// TIA Portal project "PalettizerKontrolUygulamasi" (V17)
// Vorlageprojekt für das Buch mit Zielsystem S7-1200

(* hardware
DEVICE "S7-1200-Station_1"  S7-1200 Station
   slot 0: "Baugruppenträger_0"  Rack  V1.0
   slot 1: "PLC_1"  CPU 1211C DC/DC/DC  6ES7 211-1AE40-0XB0  V4.1
*)

// ===== PLC "PLC_1"  CPU 1211C DC/DC/DC =====

VAR_GLOBAL   // PLC tag table "Standard-Variablentabelle"
   "Tag_1" AT %A0.0 : Bool;
   "Tag_2" AT %E0.0 : Bool;
   "Tag_3" AT %E0.1 : Bool;
   "AUTO" AT %I1.4 : Bool;
   "START" AT %I1.0 : Bool;
   "START LIGHT" AT %Q1.5 : Bool;
   "WARNİNG LIGHT" AT %Q1.4 : Bool;
   "BOX FEEDER" AT %Q0.6 : Bool;
   "LOAD BELT" AT %Q1.1 : Bool;
   "STOP LIGHT" AT %Q1.7 : Bool;
   "COUNTER" AT %QD30 : DWord;
   "BOX AT ENTRY" AT %I0.3 : Bool;
   "Tag_6" AT %M0.0 : Bool;
   "Tag_4" AT %QD40 : DWord;
   "Tag_5" AT %M10.0 : Bool;
   "Tag_7" AT %M10.1 : Bool;
   "ELEVATOR DOWN" AT %Q0.5 : Bool;
   "PUSH" AT %Q1.0 : Bool;
   "PUSHER LİMİT" AT %I0.4 : Bool;
   "Tag_9" AT %M0.3 : Bool;
   "Tag_8" AT %M10.6 : Bool;
   "ELEVATOR UP" AT %Q0.4 : Bool;
   "EXİT CONVEYOR" AT %Q0.2 : Bool;
   "MOVE TO LİMİT" AT %Q0.3 : Bool;
   "Tag_10" AT %M0.4 : Bool;
   "CLAMP" AT %Q1.2 : Bool;
   "Tag_12" AT %M10.2 : Bool;
   "CLAMPED" AT %I0.6 : Bool;
   "OPEN PLATE" AT %Q1.3 : Bool;
   "Tag_14" AT %M10.3 : Bool;
   "Tag_11" AT %M10.5 : Bool;
   "PLATE LİMİT" AT %I0.5 : Bool;
   "Tag_15" AT %M0.7 : Bool;
   "Tag_13" AT %M10.4 : Bool;
   "TURN" AT %Q0.7 : Bool;
   "Tag_16" AT %M1.1 : Bool;
   "Tag_17" AT %M10.7 : Bool;
   "Tag_18" AT %M1.2 : Bool;
   "Tag_19" AT %M11.0 : Bool;
   "Tag_20" AT %M11.1 : Bool;
   "Tag_21" AT %M1.3 : Bool;
   "Tag_22" AT %QD50 : DInt;
END_VAR

// folder: System blocks/Program resources

DATA_BLOCK "IEC_Timer_0_DB"   // DB1
{ S7_Optimized_Access := 'TRUE' }
AUTHOR : Simatic
FAMILY : IEC
NAME : IEC_TMR
VERSION : 1.0
// stored: InstanceOfName IEC_TIMER
"IEC_TIMER"
BEGIN
END_DATA_BLOCK

DATA_BLOCK "IEC_Timer_0_DB_1"   // DB2
{ S7_Optimized_Access := 'TRUE' }
AUTHOR : Simatic
FAMILY : IEC
NAME : IEC_TMR
VERSION : 1.0
// stored: InstanceOfName IEC_TIMER
"IEC_TIMER"
BEGIN
END_DATA_BLOCK

DATA_BLOCK "IEC_Timer_0_DB_2"   // DB3
{ S7_Optimized_Access := 'TRUE' }
AUTHOR : Simatic
FAMILY : IEC
NAME : IEC_TMR
VERSION : 1.0
// stored: InstanceOfName IEC_TIMER
"IEC_TIMER"
BEGIN
END_DATA_BLOCK

DATA_BLOCK "IEC_Timer_0_DB_3"   // DB4
{ S7_Optimized_Access := 'TRUE' }
AUTHOR : Simatic
FAMILY : IEC
NAME : IEC_TMR
VERSION : 1.0
// stored: InstanceOfName IEC_TIMER
"IEC_TIMER"
BEGIN
END_DATA_BLOCK

// folder: (top level)

FUNCTION "MHJ-PLC-Lab-Function-S71200" : Void   // FC9000, SCL
{ S7_Optimized_Access := 'TRUE' }
VERSION : 0.1
   VAR_TEMP
      rdTimeReturn : Int;
      outputTime : DTL;
      SyncVal : Byte;
      forVal : Int;
      forVal_2 : Int;
      Value : Byte;
   END_VAR
   VAR CONSTANT
      CompVal : Byte := 16#34;
      Value_01 : Byte := 16#11;
      Value_01_DW : DWord := 16#A165_D992;
      Value_02_DW : DWord := 16#58BE_4401;
   END_VAR
BEGIN

   #Value:=PEEK(area := 16#82,
        dbNumber := 0,
        byteOffset := 511);
   #Value := #Value + 1;

   POKE(area := 16#82,
        dbNumber := 0,
        byteOffset := 511,
        value := #Value);

   POKE(area:=16#81,
        dbNumber:=0,
        byteOffset:=1016,
        value:=#Value_01_DW);
   POKE(area := 16#81,
        dbNumber := 0,
        byteOffset := 1020,
        value := #Value_02_DW);

   POKE(area := 16#81,
        dbNumber := 0,
        byteOffset := 511,
        value := B#16#00);

   FOR #forVal := 0 TO 120 DO
       FOR #forVal_2:=0 TO 10 DO
           #rdTimeReturn:=RD_SYS_T(#outputTime);
           #rdTimeReturn := WR_SYS_T(#outputTime);
           #rdTimeReturn := RD_SYS_T(#outputTime);
           #rdTimeReturn := WR_SYS_T(#outputTime);
       END_FOR;
       #SyncVal:= PEEK(area := 16#81,
                      dbNumber := 0,
                      byteOffset := 511);
       IF #SyncVal = #CompVal THEN
          GOTO M_1;
       END_IF;
   END_FOR;
   RETURN;

   M_1:
   POKE(area := 16#81,
        dbNumber := 0,
        byteOffset := 511,
        value := B#16#0);
END_FUNCTION

ORGANIZATION_BLOCK "Main"   // OB1, LAD, ProgramCycle
TITLE = "Main Program Sweep (Cycle)"
{ S7_Optimized_Access := 'TRUE' }
VERSION : 0.1
   VAR_INPUT
      Initial_Call : Bool;   // Initial call of this OB
      Remanence : Bool;   // =True, if remanent data are available
   END_VAR
   VAR_TEMP   // added for the SCL form of the ladder/FBD networks
      _w1 : Bool;
      _w2 : Bool;
      _w3 : Bool;
      _w4 : Bool;
      _w5 : Bool;
      _w6 : Bool;
      _w7 : Bool;
      _w8 : Bool;
      _w9 : Bool;
      _w10 : Bool;
      _w11 : Bool;
      _w12 : Bool;
      _w13 : Bool;
   END_VAR
BEGIN

REGION Network 1: Konnektierungsbaustein für PLC-Lab
   // Im Netzwerk 1 wird der Konnektierungsbaustein für PLC-Lab aufgerufen.
   // Dieser Aufruf darf nicht entfernt werden!
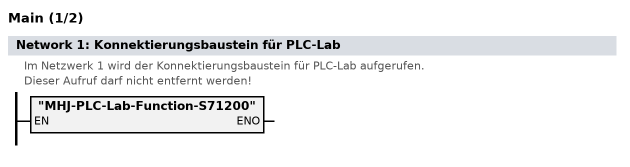
   RUNG wire#powerrail
      "MHJ-PLC-Lab-Function-S71200"()
   END_RUNG
   // the same network as SCL:
   "MHJ-PLC-Lab-Function-S71200"();
END_REGION

REGION Network 2: Ihr Programm
   // Schreiben Sie ab Netzwerk 2 Ihr Programm
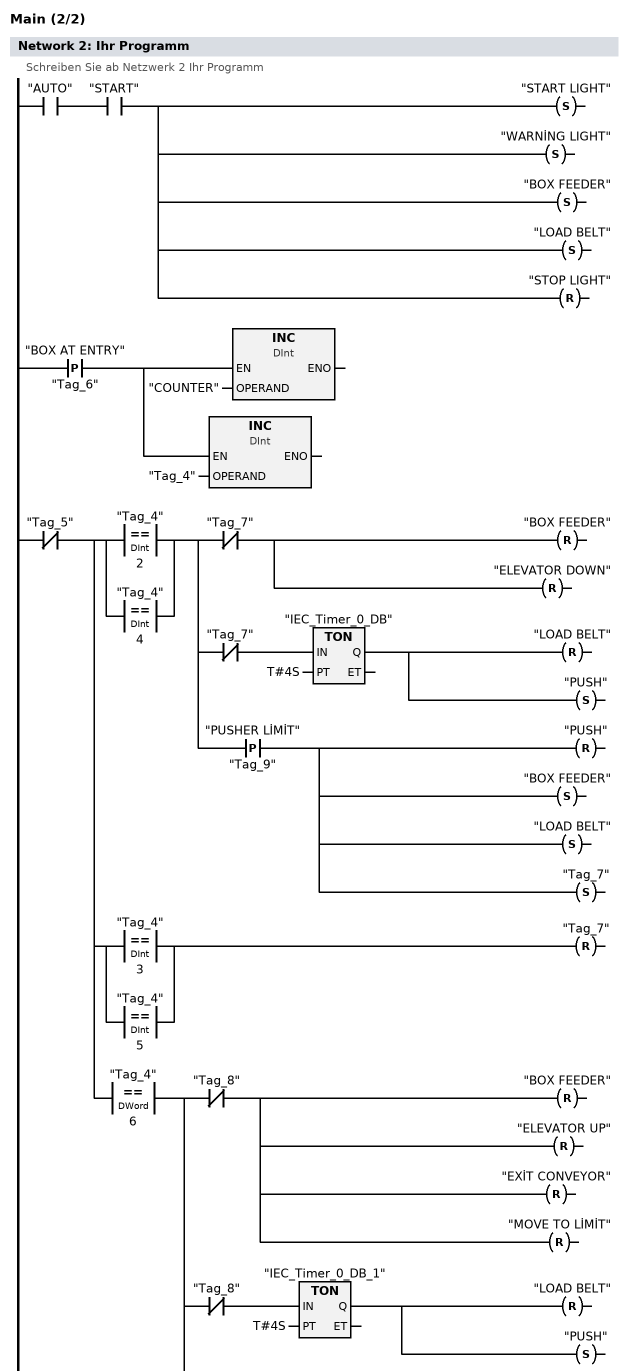
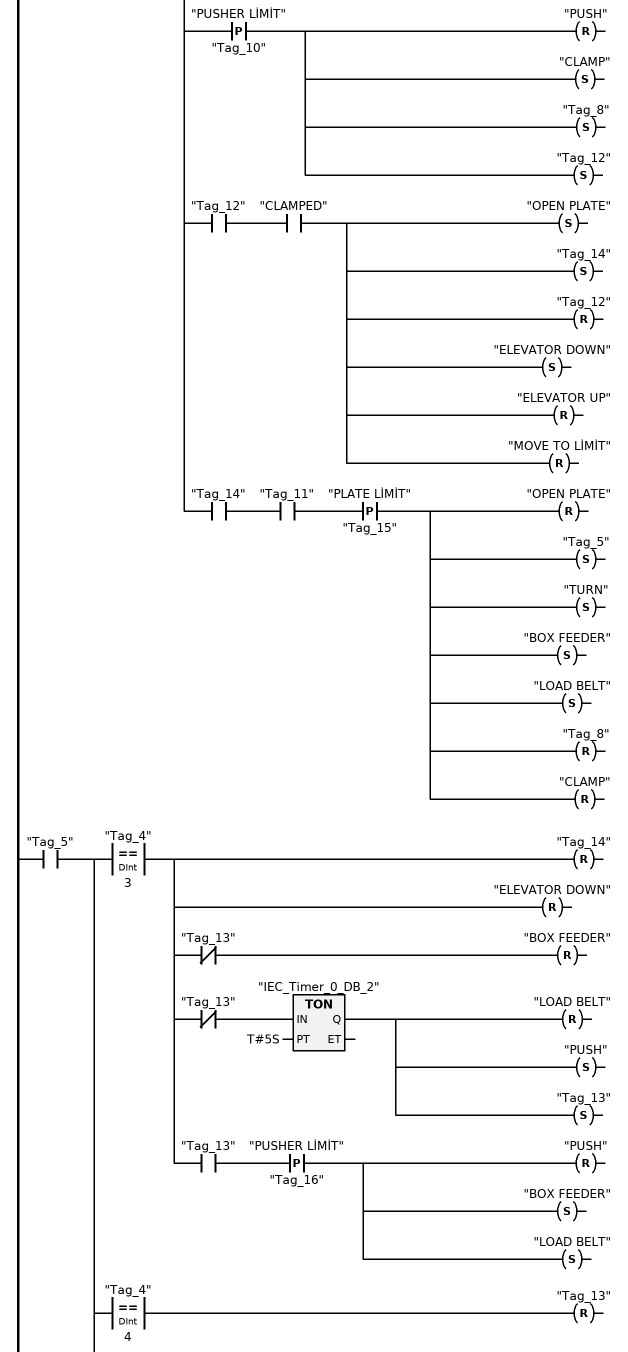
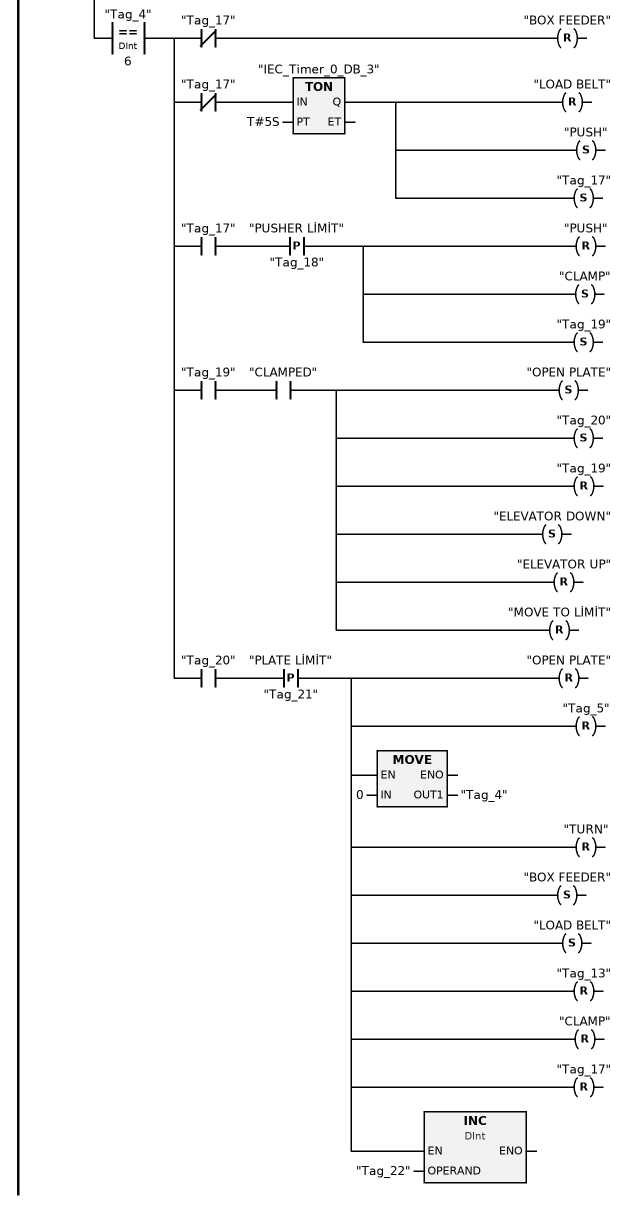
   IF "AUTO" AND "START" THEN
       "START LIGHT" := TRUE;
       "WARNİNG LIGHT" := TRUE;
       "BOX FEEDER" := TRUE;
       "LOAD BELT" := TRUE;
       "STOP LIGHT" := FALSE;
   END_IF;
   #_w1 := "BOX AT ENTRY" AND NOT "Tag_6";   // rising edge of "BOX AT ENTRY"
   "Tag_6" := "BOX AT ENTRY";
   IF #_w1 THEN
       "COUNTER" := "COUNTER" + 1;
       "Tag_4" := "Tag_4" + 1;
   END_IF;
   #_w2 := NOT "Tag_5" AND (("Tag_4" = 2) OR ("Tag_4" = 4));
   IF #_w2 AND NOT "Tag_7" THEN
       "BOX FEEDER" := FALSE;
       "ELEVATOR DOWN" := FALSE;
   END_IF;
   "IEC_Timer_0_DB".TON(IN := #_w2 AND NOT "Tag_7", PT := T#4S);
   IF "IEC_Timer_0_DB".Q THEN
       "LOAD BELT" := FALSE;
       "PUSH" := TRUE;
   END_IF;
   #_w3 := #_w2 AND "PUSHER LİMİT" AND NOT "Tag_9";   // rising edge of "PUSHER LİMİT"
   "Tag_9" := "PUSHER LİMİT";
   IF #_w3 THEN
       "PUSH" := FALSE;
       "BOX FEEDER" := TRUE;
       "LOAD BELT" := TRUE;
       "Tag_7" := TRUE;
   END_IF;
   IF NOT "Tag_5" AND (("Tag_4" = 3) OR ("Tag_4" = 5)) THEN "Tag_7" := FALSE; END_IF;
   #_w4 := NOT "Tag_5" AND ("Tag_4" = 6);
   IF #_w4 AND NOT "Tag_8" THEN
       "BOX FEEDER" := FALSE;
       "ELEVATOR UP" := FALSE;
       "EXİT CONVEYOR" := FALSE;
       "MOVE TO LİMİT" := FALSE;
   END_IF;
   "IEC_Timer_0_DB_1".TON(IN := #_w4 AND NOT "Tag_8", PT := T#4S);
   IF "IEC_Timer_0_DB_1".Q THEN
       "LOAD BELT" := FALSE;
       "PUSH" := TRUE;
   END_IF;
   #_w5 := #_w4 AND "PUSHER LİMİT" AND NOT "Tag_10";   // rising edge of "PUSHER LİMİT"
   "Tag_10" := "PUSHER LİMİT";
   IF #_w5 THEN
       "PUSH" := FALSE;
       "CLAMP" := TRUE;
       "Tag_8" := TRUE;
       "Tag_12" := TRUE;
   END_IF;
   IF #_w4 AND "Tag_12" AND "CLAMPED" THEN
       "OPEN PLATE" := TRUE;
       "Tag_14" := TRUE;
   END_IF;
   #_w6 := #_w4 AND "Tag_12" AND "CLAMPED";
   IF #_w6 THEN
       "Tag_12" := FALSE;
       "ELEVATOR DOWN" := TRUE;
       "ELEVATOR UP" := FALSE;
       "MOVE TO LİMİT" := FALSE;
   END_IF;
   #_w7 := #_w4 AND "Tag_14" AND "Tag_11" AND "PLATE LİMİT" AND NOT "Tag_15";   // rising edge of "PLATE LİMİT"
   "Tag_15" := "PLATE LİMİT";
   IF #_w7 THEN
       "OPEN PLATE" := FALSE;
       "Tag_5" := TRUE;
       "TURN" := TRUE;
       "BOX FEEDER" := TRUE;
       "LOAD BELT" := TRUE;
       "Tag_8" := FALSE;
       "CLAMP" := FALSE;
   END_IF;
   #_w8 := "Tag_5" AND ("Tag_4" = 3);
   IF #_w8 THEN
       "Tag_14" := FALSE;
       "ELEVATOR DOWN" := FALSE;
   END_IF;
   IF #_w8 AND NOT "Tag_13" THEN "BOX FEEDER" := FALSE; END_IF;
   "IEC_Timer_0_DB_2".TON(IN := #_w8 AND NOT "Tag_13", PT := T#5S);
   IF "IEC_Timer_0_DB_2".Q THEN
       "LOAD BELT" := FALSE;
       "PUSH" := TRUE;
       "Tag_13" := TRUE;
   END_IF;
   #_w9 := #_w8 AND "Tag_13" AND "PUSHER LİMİT" AND NOT "Tag_16";   // rising edge of "PUSHER LİMİT"
   "Tag_16" := "PUSHER LİMİT";
   IF #_w9 THEN
       "PUSH" := FALSE;
       "BOX FEEDER" := TRUE;
       "LOAD BELT" := TRUE;
   END_IF;
   IF "Tag_5" AND ("Tag_4" = 4) THEN "Tag_13" := FALSE; END_IF;
   #_w10 := "Tag_5" AND ("Tag_4" = 6);
   IF #_w10 AND NOT "Tag_17" THEN "BOX FEEDER" := FALSE; END_IF;
   "IEC_Timer_0_DB_3".TON(IN := #_w10 AND NOT "Tag_17", PT := T#5S);
   IF "IEC_Timer_0_DB_3".Q THEN
       "LOAD BELT" := FALSE;
       "PUSH" := TRUE;
       "Tag_17" := TRUE;
   END_IF;
   #_w11 := #_w10 AND "Tag_17" AND "PUSHER LİMİT" AND NOT "Tag_18";   // rising edge of "PUSHER LİMİT"
   "Tag_18" := "PUSHER LİMİT";
   IF #_w11 THEN
       "PUSH" := FALSE;
       "CLAMP" := TRUE;
       "Tag_19" := TRUE;
   END_IF;
   IF #_w10 AND "Tag_19" AND "CLAMPED" THEN
       "OPEN PLATE" := TRUE;
       "Tag_20" := TRUE;
   END_IF;
   #_w12 := #_w10 AND "Tag_19" AND "CLAMPED";
   IF #_w12 THEN
       "Tag_19" := FALSE;
       "ELEVATOR DOWN" := TRUE;
       "ELEVATOR UP" := FALSE;
       "MOVE TO LİMİT" := FALSE;
   END_IF;
   #_w13 := #_w10 AND "Tag_20" AND "PLATE LİMİT" AND NOT "Tag_21";   // rising edge of "PLATE LİMİT"
   "Tag_21" := "PLATE LİMİT";
   IF #_w13 THEN
       "OPEN PLATE" := FALSE;
       "Tag_5" := FALSE;
       "Tag_4" := 0;
       "TURN" := FALSE;
       "BOX FEEDER" := TRUE;
       "LOAD BELT" := TRUE;
       "Tag_13" := FALSE;
       "CLAMP" := FALSE;
       "Tag_17" := FALSE;
       "Tag_22" := "Tag_22" + 1;
   END_IF;
END_REGION
END_ORGANIZATION_BLOCK